FUNCTION_BLOCK HNLT_CN_Linkage
VAR_INPUT
	bSetStatusOn_HeatPump : BOOL;
	bAlgorithmPermission_HNLT : BOOL;
	bAlgorithmPermission_CN : BOOL;
END_VAR
VAR_OUTPUT
END_VAR
VAR
	HeatPumpSystem : FB_HeatPumpSystem;
	
	//internal variables
	bAlgorithmPermission : BOOL;
END_VAR

//check for algorithm permission
bAlgorithmPermission := bAlgorithmPermission_CN AND bAlgorithmPermission_HNLT;

//NOTE: heat pump systems contains only two-point actors -> fSetPointAutomatic = 0	
HeatPumpSystem(bSetStatusOnAutomatic := bSetStatusOn_HeatPump,
	bAlgorithmPermission := bAlgorithmPermission,
	fSetPointAutomatic := 0);

END_FUNCTION_BLOCK

(* stored: Version 1.1.0.1, ProductVersion 3.1.4024.10
   POU HNLT_CN_Linkage: Id {49b9fb4a-ee7f-4dd8-8511-b340abe8c57d}, SpecialFunc None *)
